Universal Robots PolyScope program: cognex02.urp

Program cognex02 (installation=default directory=/programs createdIn=5.9.1.1031110 lastSavedIn=5.9.1.1031110 robotSerialNumber=20195501059)
Calibrated DH parameters: a=[0.000146, -0.418764, -0.053981, 0.000058, -0.000023, 0]; d=[0.162545, 37.319448, -206.067439, 168.881546, 0.09955, 0.099464]; alpha=[1.57004, -0.001979, 0.002304, 1.570607, -1.57066, 0]; deltaTheta=[0, -0.174616, -1.258233, 1.432844, -0.000001, 0]
Robot Program (runOnlyOnce=true)
  MoveJ speed 60 deg/s, acceleration 80 deg/s^2 (useActiveTCP=true) feature=Base
    Waypoint inspect_p: TCP in base x=256.42 y=-582.871 z=37.895 mm, rx=1.7053 ry=1.7139 rz=-0.7255 rad; joints [105.659, -56.488, 127.219, -208.303, 260.641, -258.656] deg; TCP offset x=0 y=0 z=174 mm, rx=0 ry=0 rz=0 rad
  URCap Cognex Camera Pose (Cognex In-Sight Robot Guidance, Cognex Corporation) dataModel(newNode=false, rotLock=true, btnClearRef=true, Pose(key=refPose, Position(key=posePosition, Length(key=X value=0.256384 unit=M), Length(key=Y value=-0.665024 unit=M), Length(key=Z value=0.037922 unit=M)), Rotation(key=poseRotation, Angle(key=RX value=1.705286 unit=RAD), Angle(key=RY value=1.713874 unit=RAD), Angle(key=RZ value=-0.725574 unit=RAD))), Variable(key=selectedVar, variable(name=CGX_result)))
    URCap Job Pass (Cognex In-Sight Robot Guidance, Cognex Corporation)
      MoveL speed 250 mm/s, acceleration 1200 mm/s^2 (useActiveTCP=true) feature=Base
        Waypoint Waypoint (Variable): variable=CGX_result
      URCap Cognex Camera Pose (Cognex In-Sight Robot Guidance, Cognex Corporation) dataModel(newNode=false, rotLock=true, btnClearRef=true, camMount=true, Variable(key=selectedVar, variable(name=CGX_result_1)), Pose(key=refPose, Position(key=posePosition, Length(key=X value=0.256426 unit=M), Length(key=Y value=-0.582864 unit=M), Length(key=Z value=0.037873 unit=M)), Rotation(key=poseRotation, Angle(key=RX value=1.705252 unit=RAD), Angle(key=RY value=1.713976 unit=RAD), Angle(key=RZ value=-0.725469 unit=RAD))))
        URCap Job Pass (Cognex In-Sight Robot Guidance, Cognex Corporation)
          MoveL speed 250 mm/s, acceleration 1200 mm/s^2 (useActiveTCP=true) feature=Base
            Waypoint Waypoint (Variable): variable=CGX_result_1
        URCap Job Fail (Cognex In-Sight Robot Guidance, Cognex Corporation)
          'ttt'
        URCap No Response (Cognex In-Sight Robot Guidance, Cognex Corporation)
          'yyy'
    URCap Job Fail (Cognex In-Sight Robot Guidance, Cognex Corporation)
      Popup Message (haltProgram=false message=fail inputType=Text)
    URCap No Response (Cognex In-Sight Robot Guidance, Cognex Corporation)
      Popup Message (haltProgram=false message=no response inputType=Text)
  MoveL speed 250 mm/s, acceleration 1200 mm/s^2 (useActiveTCP=true) feature=Base
    Waypoint inspect_p: TCP in base x=256.42 y=-582.871 z=37.895 mm, rx=1.7053 ry=1.7139 rz=-0.7255 rad; joints [105.659, -56.488, 127.219, -208.303, 260.641, -258.656] deg
